{attribute 'qualified_only'}
VAR_GLOBAL
END_VAR

(* stored: Version 1.1.0.1, ProductVersion 3.1.4022.7
   GVL GVL_04_Auto_Servo_Motor: Id {61133314-e00d-4b37-8afa-b981004a9b52} *)
